(* CODESYS project EtherNet.multinode190308.3.project

Project tree, tasks and I/O mapping:
  MIC7001_A : Changsha-Cyber-MI-linux, Changsha Cyber-MI Co., Ltd., version 3.5.10.40
    application Application
      libraries: Standard, * (System); SysFile, 3.5.9.0 (System); SysTypes2 Interfaces, * (System); SysShm, * (System); CAA Mathematics, * (CAA Technical Workgroup); CAA Net Base Services, * (CAA Technical Workgroup); SysTime, 3.5.9.0 (System); CAA Types Extern, 3.5.10.0 (CAA Technical Workgroup)
      task c_MainTask (cyclic, interval 20 ms, priority 15) calls prg_ethernet
      data type STATE
      programs/
        program prg_ethernet [ST]
      funcs/
        function fn_set_ip [ST]
        function fn_read_ip [ST]
      global variables GVL
    SoftMotion General Axis Pool
  MIC7001_B : Changsha-Cyber-MI-linux, Changsha Cyber-MI Co., Ltd., version 3.5.10.40
    application Application
      libraries: Standard, * (System); SysFile, 3.5.9.0 (System); SysTypes2 Interfaces, * (System); SysShm, * (System); CAA Mathematics, * (CAA Technical Workgroup); CAA Net Base Services, * (CAA Technical Workgroup); SysTime, 3.5.9.0 (System); CAA Types Extern, 3.5.10.0 (CAA Technical Workgroup)
      task c_MainTask (cyclic, interval 20 ms, priority 15) calls prg_ethernet
      programs/
        program prg_ethernet [ST]
      data type STATE
      funcs/
        function fn_set_ip [ST]
        function fn_read_ip [ST]
      global variables GVL
    SoftMotion General Axis Pool
  MIC7001_C : Changsha-Cyber-MI-linux, Changsha Cyber-MI Co., Ltd., version 3.5.10.40
    application Application
      libraries: Standard, * (System); SysFile, 3.5.9.0 (System); SysTypes2 Interfaces, * (System); SysShm, * (System); CAA Mathematics, * (CAA Technical Workgroup); CAA Net Base Services, * (CAA Technical Workgroup); SysTime, 3.5.9.0 (System); CAA Types Extern, 3.5.10.0 (CAA Technical Workgroup)
      task c_MainTask (cyclic, interval 20 ms, priority 15) calls prg_ethernet
      programs/
        program prg_ethernet [ST]
      data type STATE
      funcs/
        function fn_set_ip [ST]
        function fn_read_ip [ST]
      global variables GVL
    SoftMotion General Axis Pool
  libraries: VisuSymbols, 3.5.10.0 (System)
  5ce3da45-db07-42e7-a21c-a00fff4ed8f6|C:\Users\zhou\p01.bmp
  5ce3da45-db07-42e7-a21c-a00fff4ed8f6|C:\working\p01.bmp
  5ce3da45-db07-42e7-a21c-a00fff4ed8f6|C:\working\file.bmp
  text list GlobalTextList
*)

// MIC7001_A/Application/STATE
TYPE STATE :
(
	INIT := 0, 	(* first State. Connections are set up *)
	SEND,		(* Send messages *)
	RECV,		(* Receive messages *)
	ERROR		(* Prepare to reset connections *)
);
END_TYPE

// MIC7001_B/Application/STATE
TYPE STATE :
(
	INIT := 0, 	(* first State. Connections are set up *)
	SEND,		(* Send messages *)
	RECV,		(* Receive messages *)
	ERROR		(* Prepare to reset connections *)
);
END_TYPE

// MIC7001_C/Application/STATE
TYPE STATE :
(
	INIT := 0, 	(* first State. Connections are set up *)
	SEND,		(* Send messages *)
	RECV,		(* Receive messages *)
	ERROR		(* Prepare to reset connections *)
);
END_TYPE

// MIC7001_A/Application/GVL
{attribute 'qualified_only'}
VAR_GLOBAL
	ipaddr:STRING := '192.168.1.251';   //设置本设备的IP地址，几台设备在同一网段，即： 只修改前面的最后一段（251）
	recv_port:UINT := 15001;  //本设备发送端口号
	send_port:UINT := 15002;  //本设备接收端口号
	
	g_send_flag :BOOL := FALSE;  //发送命令，为 true则启动一次发送，完成后清除标志
	g_buf_send:ARRAY[0..255] OF BYTE;  //发送缓冲区
	g_buf_recv:ARRAY[0..255] OF BYTE;  //接收缓冲区
END_VAR

// MIC7001_B/Application/GVL
{attribute 'qualified_only'}
VAR_GLOBAL
	ipaddr:STRING := '192.168.1.252';   //设置本设备的IP地址，几台设备在同一网段，即： 只修改前面的最后一段（252）
	recv_port:UINT := 15001;  //本设备发送端口号
	send_port:UINT := 15002;  //本设备接收端口号
	
	g_send_flag :BOOL := FALSE;  //发送命令，为 true则启动一次发送，完成后清除标志
	g_buf_send:ARRAY[0..255] OF BYTE;  //发送缓冲区
	g_buf_recv:ARRAY[0..255] OF BYTE;  //接收缓冲区
END_VAR

// MIC7001_C/Application/GVL
{attribute 'qualified_only'}
VAR_GLOBAL
	ipaddr:STRING := '192.168.1.253';   //设置本设备的IP地址，几台设备在同一网段，即： 只修改前面的最后一段（253）
	recv_port:UINT := 15001;  //本设备发送端口号
	send_port:UINT := 15002;  //本设备接收端口号
	
	g_send_flag :BOOL := FALSE;  //发送命令，为 true则启动一次发送，完成后清除标志
	g_buf_send:ARRAY[0..255] OF BYTE;  //发送缓冲区
	g_buf_recv:ARRAY[0..255] OF BYTE;  //接收缓冲区
END_VAR

// MIC7001_A/Application/programs/prg_ethernet
PROGRAM prg_ethernet
VAR  
	eSTATE		: STATE; (* 状态转换变量 *)
	myIP		: NBS.IP_ADDR; (* MIC7001本身的IP地址 *)
	myPort		: UINT; (* MIC7001用于通信的端口 *)
	IPSend		: NBS.IP_ADDR ; (* 对方的IP地址 *)
	PortSend	: UINT ; (* 对方的端口 *)

	ctRecAnswers	: CAA.COUNT; (* No. of received messages *)
	ctSentMessage	: CAA.COUNT; (* No. of sent messages *)
	ctErrorCounter	: CAA.COUNT; (* No. connection errors *)

	UDPPeer			: NBS.UDP_Peer; (* FB UDP Peer *)
	UDPSend			: NBS.UDP_Send; (* FB UDP Send *)
	UDPReceive		: NBS.UDP_Receive; (* FB UDP Receive *)
	
	Peer			: CAA.HANDLE; (* Handle to the peer connection *)
	
	/// 辅助变量 
	i				: UINT;
	sTmp1			: STRING;
	xEnable			: BOOL;
	
	ipstr:STRING(32);
END_VAR


CASE eSTATE OF

STATE.INIT:  //初始化状态
	IF NOT fn_read_ip(ADR(ipstr)) OR ipstr <> gvl.ipaddr THEN   //读取原有的IP地址，如果与本程序中设置的不同，则自动更改(更改后需要重启生效）
		ipstr := gvl.ipaddr;
		fn_set_ip(ADR(ipstr), len(ipstr));
	END_IF 

	myIP.sAddr:= gvl.ipaddr;	
	myPort:= gvl.recv_port;
	
	xEnable:= TRUE;  //用于启动下面最后一行的UDPPeer功能块
	// 建立连接后马上转到接收状态
	IF UDPPeer.xActive THEN 
		eSTATE:= STATE.RECV;
	ELSIF UDPPeer.xError THEN
		eSTATE:= STATE.ERROR;
	END_IF

	gvl.g_buf_send[0] := 16#41;
	gvl.g_buf_send[1] := 16#42;
	gvl.g_buf_send[2] := 16#43;
	gvl.g_buf_send[3] := 16#44;
	
STATE.RECV:  //接收状态
	//如果出现错误，进入错误状态
	IF UDPPeer.xActive THEN 
		UDPReceive(xEnable:= TRUE,  hPeer:= Peer, szSize:= SIZEOF(gvl.g_buf_recv), pData:= ADR(gvl.g_buf_recv));
		IF UDPReceive.xReady THEN
			ctRecAnswers:= ctRecAnswers +1;
			gvl.g_send_flag := TRUE;
		ELSIF UDPReceive.xError THEN
			eSTATE:= STATE.ERROR;
		END_IF
	ELSE
		eSTATE:= STATE.ERROR;
	END_IF
	
	IF gvl.g_send_flag THEN
		eSTATE:= STATE.SEND;
		UDPSend(xExecute:= FALSE);	//发送之前初始化发送功能块
	END_IF
	
STATE.SEND:  //发送状态
	//发送一个字符串加一个数字（100到0）
	IF UDPPeer.xActive THEN 
		//发送数据到 MIC7001_B
		IPSend.sAddr := '192.168.1.222';	
		PortSend := 15601;
		UDPSend(xExecute:= TRUE, udiTimeOut:= 0, hPeer:= Peer, ipAddr:= IPSend, uiPort:= PortSend, szSize:= SIZEOF(gvl.g_buf_send), pData:= ADR(gvl.g_buf_send));
		
		//发送数据到MIC7001_C
		IPSend.sAddr := '192.168.1.253';	
		PortSend := 15002;
		UDPSend(xExecute:= TRUE, udiTimeOut:= 0, hPeer:= Peer, ipAddr:= IPSend, uiPort:= PortSend, szSize:= SIZEOF(gvl.g_buf_send), pData:= ADR(gvl.g_buf_send));	
	
		//发送成功后转入接收状态
		IF UDPSend.xDone THEN 
			UDPSend(xExecute:= FALSE);	//发送完成后初始化发送功能块
			gvl.g_send_flag := FALSE;
			eSTATE:= STATE.RECV;
		ELSIF UDPSend.xError THEN
			eSTATE:= STATE.ERROR;		
		END_IF
	ELSE
		eSTATE:= STATE.ERROR;
	END_IF

STATE.ERROR:  //错误状态
	ctErrorCounter:= ctErrorCounter +1;
	UDPPeer(xEnable:= FALSE, ipAddr:= myIP, uiPort:= myPort, hPeer=> Peer);
	gvl.g_send_flag := FALSE;
	eState := STATE.INIT;	 //回到初始化状态，重新开始
END_CASE

//保持每个周期调用，维护与对方的连接关系本地端口的接收状态
UDPPeer(xEnable:= xEnable, ipAddr:= myIP, uiPort:= myPort, hPeer=> Peer);

END_PROGRAM

// MIC7001_A/Application/funcs/fn_read_ip
FUNCTION fn_read_ip : BOOL
VAR_INPUT
	ip: POINTER TO STRING;
END_VAR

VAR
	hFile: RTS_IEC_HANDLE;
	udiOpenError: RTS_IEC_RESULT;
	udiReadError: RTS_IEC_RESULT;
	i :INT;
	iTemp: UDINT;
	udiPos: UDINT;
	str_size: __XWORD;
	udiByteRead: LWORD;

	len_of_line: INT;
	len_of_number :INT;
	magicNumber:REAL;
	check_sum:REAL:= 0;
	temp_num:REAL;
END_VAR

fn_read_ip := FALSE;

//检测文件是否存在
hFile := sysfileopen(szFile := '/userapp/ipaddr.txt', am := sysfile.AM_READ, pResult:= ADR(udiOpenError));
IF hFile = RTS_INVALID_HANDLE	THEN  //文件不存在
	RETURN;
END_IF
//文件存在，开始读取内容
udiPos := SysFileSetPos(hFile:=hFile, ulOffset := 0);
udiByteRead := sysfile.SysFileRead(hfile := hFile,pbyBuffer := ip, ulSize := 32, pResult := ADR(udiReadError));
IF udiByteRead < 4 THEN  //读取失败
	sysfile.SysFileClose(hFile := hFile);
	RETURN;
END_IF

fn_read_ip := TRUE;

END_FUNCTION

// MIC7001_B/Application/funcs/fn_read_ip
FUNCTION fn_read_ip : BOOL
VAR_INPUT
	ip: POINTER TO STRING;
END_VAR

VAR
	hFile: RTS_IEC_HANDLE;
	udiOpenError: RTS_IEC_RESULT;
	udiReadError: RTS_IEC_RESULT;
	i :INT;
	iTemp: UDINT;
	udiPos: UDINT;
	str_size: __XWORD;
	udiByteRead: LWORD;

	len_of_line: INT;
	len_of_number :INT;
	magicNumber:REAL;
	check_sum:REAL:= 0;
	temp_num:REAL;
END_VAR

fn_read_ip := FALSE;

//检测文件是否存在
hFile := sysfileopen(szFile := '/userapp/ipaddr.txt', am := sysfile.AM_READ, pResult:= ADR(udiOpenError));
IF hFile = RTS_INVALID_HANDLE	THEN  //文件不存在
	RETURN;
END_IF
//文件存在，开始读取内容
udiPos := SysFileSetPos(hFile:=hFile, ulOffset := 0);
udiByteRead := sysfile.SysFileRead(hfile := hFile,pbyBuffer := ip, ulSize := 32, pResult := ADR(udiReadError));
IF udiByteRead < 4 THEN  //读取失败
	sysfile.SysFileClose(hFile := hFile);
	RETURN;
END_IF

fn_read_ip := TRUE;

END_FUNCTION

// MIC7001_C/Application/funcs/fn_read_ip
FUNCTION fn_read_ip : BOOL
VAR_INPUT
	ip: POINTER TO STRING;
END_VAR

VAR
	hFile: RTS_IEC_HANDLE;
	udiOpenError: RTS_IEC_RESULT;
	udiReadError: RTS_IEC_RESULT;
	i :INT;
	iTemp: UDINT;
	udiPos: UDINT;
	str_size: __XWORD;
	udiByteRead: LWORD;

	len_of_line: INT;
	len_of_number :INT;
	magicNumber:REAL;
	check_sum:REAL:= 0;
	temp_num:REAL;
END_VAR

fn_read_ip := FALSE;

//检测文件是否存在
hFile := sysfileopen(szFile := '/userapp/ipaddr.txt', am := sysfile.AM_READ, pResult:= ADR(udiOpenError));
IF hFile = RTS_INVALID_HANDLE	THEN  //文件不存在
	RETURN;
END_IF
//文件存在，开始读取内容
udiPos := SysFileSetPos(hFile:=hFile, ulOffset := 0);
udiByteRead := sysfile.SysFileRead(hfile := hFile,pbyBuffer := ip, ulSize := 32, pResult := ADR(udiReadError));
IF udiByteRead < 4 THEN  //读取失败
	sysfile.SysFileClose(hFile := hFile);
	RETURN;
END_IF

fn_read_ip := TRUE;

END_FUNCTION

// MIC7001_A/Application/funcs/fn_set_ip
FUNCTION fn_set_ip : BOOL
VAR_INPUT
	ip: POINTER TO STRING;
	len:DINT;
END_VAR
VAR
	hFile: RTS_IEC_HANDLE;
	udiOpenError: RTS_IEC_RESULT;
	udiReadError: RTS_IEC_RESULT;
	udiWriteError: RTS_IEC_RESULT;
	i :INT;
	iTemp: UDINT;
	udiPos: UDINT;
	str_size: __XWORD;
	udiByteRead: UDINT;

	len_of_line: INT;
	len_of_number :INT;
	magicNumber:REAL;
	check_sum:REAL:= 0;
	temp_num:REAL;
	udiByteWrite: LWORD;
END_VAR


fn_set_ip := FALSE;

hFile := sysfileopen(szFile := '/userapp/ipaddr.txt', am := sysfile.AM_WRITE, pResult := ADR(udiOpenError));
IF hFile = RTS_INVALID_HANDLE THEN //创建文件失败
	RETURN;
END_IF

udiPos := SysFileSetPos(hFile:=hFile, ulOffset:=0);	
udiByteWrite := sysfile.SysFileWrite(hFile := hFile,pbyBuffer := ip,ulSize := len, pResult := ADR(udiWriteError));
IF udiByteWrite = 0 THEN
	RETURN;
END_IF

fn_set_ip := TRUE;
RETURN;

END_FUNCTION

// MIC7001_B/Application/funcs/fn_set_ip
FUNCTION fn_set_ip : BOOL
VAR_INPUT
	ip: POINTER TO STRING;
	len:DINT;
END_VAR
VAR
	hFile: RTS_IEC_HANDLE;
	udiOpenError: RTS_IEC_RESULT;
	udiReadError: RTS_IEC_RESULT;
	udiWriteError: RTS_IEC_RESULT;
	i :INT;
	iTemp: UDINT;
	udiPos: UDINT;
	str_size: __XWORD;
	udiByteRead: UDINT;

	len_of_line: INT;
	len_of_number :INT;
	magicNumber:REAL;
	check_sum:REAL:= 0;
	temp_num:REAL;
	udiByteWrite: LWORD;
END_VAR


fn_set_ip := FALSE;

hFile := sysfileopen(szFile := '/userapp/ipaddr.txt', am := sysfile.AM_WRITE, pResult := ADR(udiOpenError));
IF hFile = RTS_INVALID_HANDLE THEN //创建文件失败
	RETURN;
END_IF

udiPos := SysFileSetPos(hFile:=hFile, ulOffset:=0);	
udiByteWrite := sysfile.SysFileWrite(hFile := hFile,pbyBuffer := ip,ulSize := len, pResult := ADR(udiWriteError));
IF udiByteWrite = 0 THEN
	RETURN;
END_IF

fn_set_ip := TRUE;
RETURN;

END_FUNCTION

// MIC7001_C/Application/funcs/fn_set_ip
FUNCTION fn_set_ip : BOOL
VAR_INPUT
	ip: POINTER TO STRING;
	len:DINT;
END_VAR
VAR
	hFile: RTS_IEC_HANDLE;
	udiOpenError: RTS_IEC_RESULT;
	udiReadError: RTS_IEC_RESULT;
	udiWriteError: RTS_IEC_RESULT;
	i :INT;
	iTemp: UDINT;
	udiPos: UDINT;
	str_size: __XWORD;
	udiByteRead: UDINT;

	len_of_line: INT;
	len_of_number :INT;
	magicNumber:REAL;
	check_sum:REAL:= 0;
	temp_num:REAL;
	udiByteWrite: LWORD;
END_VAR


fn_set_ip := FALSE;

hFile := sysfileopen(szFile := '/userapp/ipaddr.txt', am := sysfile.AM_WRITE, pResult := ADR(udiOpenError));
IF hFile = RTS_INVALID_HANDLE THEN //创建文件失败
	RETURN;
END_IF

udiPos := SysFileSetPos(hFile:=hFile, ulOffset:=0);	
udiByteWrite := sysfile.SysFileWrite(hFile := hFile,pbyBuffer := ip,ulSize := len, pResult := ADR(udiWriteError));
IF udiByteWrite = 0 THEN
	RETURN;
END_IF

fn_set_ip := TRUE;
RETURN;

END_FUNCTION

// MIC7001_B/Application/programs/prg_ethernet
PROGRAM prg_ethernet
VAR  
	eSTATE		: STATE; (* 状态转换变量 *)
	myIP		: NBS.IP_ADDR; (* MIC7001本身的IP地址 *)
	myPort		: UINT; (* MIC7001用于通信的端口 *)
	IPSend		: NBS.IP_ADDR ; (* 对方的IP地址 *)
	PortSend	: UINT ; (* 对方的端口 *)

	ctRecAnswers	: CAA.COUNT; (* No. of received messages *)
	ctSentMessage	: CAA.COUNT; (* No. of sent messages *)
	ctErrorCounter	: CAA.COUNT; (* No. connection errors *)

	UDPPeer			: NBS.UDP_Peer; (* FB UDP Peer *)
	UDPSend			: NBS.UDP_Send; (* FB UDP Send *)
	UDPReceive		: NBS.UDP_Receive; (* FB UDP Receive *)
	
	Peer			: CAA.HANDLE; (* Handle to the peer connection *)
	
	/// 辅助变量 
	i				: UINT;
	sTmp1			: STRING;
	xEnable			: BOOL;
	
	ipstr:STRING(32);
END_VAR


CASE eSTATE OF

STATE.INIT:  //初始化状态
	IF NOT fn_read_ip(ADR(ipstr)) OR ipstr <> gvl.ipaddr THEN   //读取原有的IP地址，如果与本程序中设置的不同，则自动更改(更改后需要重启生效）
		ipstr := gvl.ipaddr;
		fn_set_ip(ADR(ipstr), len(ipstr));
	END_IF 

	myIP.sAddr:= gvl.ipaddr;	
	myPort:= gvl.recv_port;
	
	xEnable:= TRUE;  //用于启动下面最后一行的UDPPeer功能块
	// 建立连接后马上转到接收状态
	IF UDPPeer.xActive THEN 
		eSTATE:= STATE.RECV;
	ELSIF UDPPeer.xError THEN
		eSTATE:= STATE.ERROR;
	END_IF

STATE.RECV:  //接收状态
	//如果出现错误，进入错误状态
	IF UDPPeer.xActive THEN 
		UDPReceive(xEnable:= TRUE,  hPeer:= Peer, szSize:= SIZEOF(gvl.g_buf_recv), pData:= ADR(gvl.g_buf_recv));
		IF UDPReceive.xReady THEN
			ctRecAnswers:= ctRecAnswers +1;
		ELSIF UDPReceive.xError THEN
			eSTATE:= STATE.ERROR;
		END_IF
	ELSE
		eSTATE:= STATE.ERROR;
	END_IF
	
	IF gvl.g_send_flag THEN
		eSTATE:= STATE.SEND;
		UDPSend(xExecute:= FALSE);	//发送之前初始化发送功能块
	END_IF
	
STATE.SEND:  //发送状态
	IF UDPPeer.xActive THEN 
		IPSend.sAddr := '192.168.1.251';	
		PortSend := 15001;
		UDPSend(xExecute:= TRUE, udiTimeOut:= 0, hPeer:= Peer, ipAddr:= IPSend, uiPort:= PortSend, szSize:= SIZEOF(gvl.g_buf_send), pData:= ADR(gvl.g_buf_send));
		//发送成功后转入接收状态
		IF UDPSend.xDone THEN 
			UDPSend(xExecute:= FALSE);	//发送完成后初始化发送功能块
			gvl.g_send_flag := FALSE;
			eSTATE:= STATE.RECV;
		ELSIF UDPSend.xError THEN
			eSTATE:= STATE.ERROR;		
		END_IF
	ELSE
		eSTATE:= STATE.ERROR;
	END_IF

STATE.ERROR:  //错误状态
	ctErrorCounter:= ctErrorCounter +1;
	UDPPeer(xEnable:= FALSE, ipAddr:= myIP, uiPort:= myPort, hPeer=> Peer);
	gvl.g_send_flag := FALSE;
	eState := STATE.INIT;	 //回到初始化状态，重新开始
END_CASE

//保持每个周期调用，维护与对方的连接关系本地端口的接收状态
UDPPeer(xEnable:= xEnable, ipAddr:= myIP, uiPort:= myPort, hPeer=> Peer);

END_PROGRAM

// MIC7001_C/Application/programs/prg_ethernet
PROGRAM prg_ethernet
VAR  
	eSTATE		: STATE; (* 状态转换变量 *)
	myIP		: NBS.IP_ADDR; (* MIC7001本身的IP地址 *)
	myPort		: UINT; (* MIC7001用于通信的端口 *)
	IPSend		: NBS.IP_ADDR; (* 对方的IP地址 *)
	PortSend	: UINT ; (* 对方的端口 *)

	ctRecAnswers	: CAA.COUNT; (* No. of received messages *)
	ctSentMessage	: CAA.COUNT; (* No. of sent messages *)
	ctErrorCounter	: CAA.COUNT; (* No. connection errors *)

	UDPPeer			: NBS.UDP_Peer; (* FB UDP Peer *)
	UDPSend			: NBS.UDP_Send; (* FB UDP Send *)
	UDPReceive		: NBS.UDP_Receive; (* FB UDP Receive *)
	
	Peer			: CAA.HANDLE; (* Handle to the peer connection *)
	
	/// 辅助变量 
	i				: UINT;
	sTmp1			: STRING;
	xEnable			: BOOL;
	
	ipstr:STRING(32);
END_VAR


CASE eSTATE OF

STATE.INIT:  //初始化状态
	IF NOT fn_read_ip(ADR(ipstr)) OR ipstr <> gvl.ipaddr THEN   //读取原有的IP地址，如果与本程序中设置的不同，则自动更改(更改后需要重启生效）
		ipstr := gvl.ipaddr;
		fn_set_ip(ADR(ipstr), len(ipstr));
	END_IF 

	myIP.sAddr:= gvl.ipaddr;	
	myPort:= gvl.recv_port;
	
	xEnable:= TRUE;  //用于启动下面最后一行的UDPPeer功能块
	// 建立连接后马上转到接收状态
	IF UDPPeer.xActive THEN 
		eSTATE:= STATE.RECV;
	ELSIF UDPPeer.xError THEN
		eSTATE:= STATE.ERROR;
	END_IF

STATE.RECV:  //接收状态
	//如果出现错误，进入错误状态
	IF UDPPeer.xActive THEN 
		UDPReceive(xEnable:= TRUE,  hPeer:= Peer, szSize:= SIZEOF(gvl.g_buf_recv), pData:= ADR(gvl.g_buf_recv));
		IF UDPReceive.xReady THEN
			ctRecAnswers:= ctRecAnswers +1;
		ELSIF UDPReceive.xError THEN
			eSTATE:= STATE.ERROR;
		END_IF
	ELSE
		eSTATE:= STATE.ERROR;
	END_IF
	
	IF gvl.g_send_flag THEN
		eSTATE:= STATE.SEND;
		UDPSend(xExecute:= FALSE);	//发送之前初始化发送功能块
	END_IF
	
STATE.SEND:  //发送状态
	IF UDPPeer.xActive THEN 
		IPSend.sAddr := '192.168.1.251';	
		PortSend := 15001;
		UDPSend(xExecute:= TRUE, udiTimeOut:= 0, hPeer:= Peer, ipAddr:= IPSend, uiPort:= PortSend, szSize:= SIZEOF(gvl.g_buf_send), pData:= ADR(gvl.g_buf_send));
		//发送成功后转入接收状态
		IF UDPSend.xDone THEN 
			UDPSend(xExecute:= FALSE);	//发送完成后初始化发送功能块
			gvl.g_send_flag := FALSE;
			eSTATE:= STATE.RECV;
		ELSIF UDPSend.xError THEN
			eSTATE:= STATE.ERROR;		
		END_IF
	ELSE
		eSTATE:= STATE.ERROR;
	END_IF

STATE.ERROR:  //错误状态
	ctErrorCounter:= ctErrorCounter +1;
	UDPPeer(xEnable:= FALSE, ipAddr:= myIP, uiPort:= myPort, hPeer=> Peer);
	gvl.g_send_flag := FALSE;
	eState := STATE.INIT;	 //回到初始化状态，重新开始
END_CASE

//保持每个周期调用，维护与对方的连接关系本地端口的接收状态
UDPPeer(xEnable:= xEnable, ipAddr:= myIP, uiPort:= myPort, hPeer=> Peer);

END_PROGRAM
